// TIA Portal V18 export
TYPE "RemConsole_IO_Out"
   STRUCT
      PTOLED : Bool;
      HPUFaultLED : Bool;
      TDFaultLED : Bool;
      BUWClLED : Bool;
      TDEnLED : Bool;
      Spare_6 : Bool;
      MSVClLED : Bool;
      QuillLockedLED : Bool;
      ElevClLED : Bool;
      Horn : Bool;
      MSVClInt : Bool;
      BUWClInt : Bool;
      Spare_7 : Bool;
      Spare_8 : Bool;
      Spare_9 : Bool;
      Spare_10 : Bool;
      Spare_11 : Bool;
      Spare_12 : Bool;
      Spare_13 : Bool;
      Spare_14 : Bool;
      Spare_15 : Bool;
      Spare : Bool;
      Spare_16 : Bool;
      Spare_17 : Bool;
      Spare_18 : Bool;
      Spare_19 : Bool;
      Spare_1 : Bool;
      Spare_2 : Bool;
      Spare_3 : Bool;
      Spare_4 : Bool;
      Spare_5 : Bool;
      Spare_20 : Bool;
      DrillRecTorq : Int;
      DrillRecRPM : Int;
      SpareAO : Int;
      SpareAO_2 : Int;
   END_STRUCT;
END_TYPE
